{attribute addProperty BoxType "EL3182-0000-0016"}
{attribute addProperty Id "Ch_1_Al_InputsCh_1_Al_Inputs_D230195D324"}
{attribute addProperty CRC "2589471246"}
{attribute addProperty SizeInBites "32"}
{attribute addProperty SizeInBytes "4"}
TYPE Ch_1_9A58320E :
STRUCT
	{attribute addProperty Name "Ch_1_Al_Inputs"}
	Ch_1_Al_Inputs  : Ch_1_Al_Inputs_D230195D;
END_STRUCT
END_TYPE

(* stored: Version 1.2.0.0, ProductVersion 3.1.4024.9
   DUT Ch_1_9A58320E: Id {79e3dc5f-3281-485b-8863-ad53bf9ab849} *)
